// ---- VISUs/HMI.TcVIS
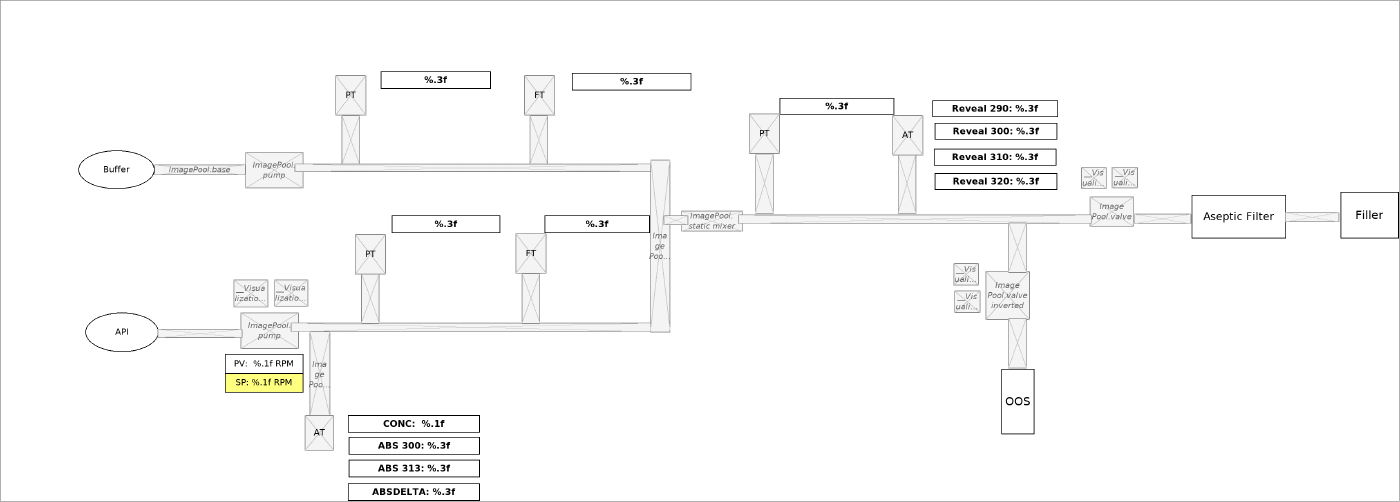
VISUALIZATION HMI  // 1787x641
    Ellipse (100,192 97x49), "Buffer"
    Ellipse (109,399 93x50), "API"
    Line (254,369)
    Line (836,413) (379,413)
    Line (449,161) (449,206)
    Line (967,273)
    Rectangle (1278,471 42x83), "OOS"
    Rectangle (1521,249 120x55), "Aseptic Filter"
    Rectangle (1711,245 74x59), "Filler"
    Image (307,399 74x46), image: ImagePool.pump
    Image (313,194 74x46), image: ImagePool.pump
    Image (869,269 79x26), image: ImagePool.static mixer
    Image (1391,251 56x38), image: ImagePool.valve
    Image (1258,346 56x62), image: ImagePool.valve inverted
    Rectangle (730,93 152x22), "%.3f", text variable: IO.FT_Buff_PV
    Rectangle (486,91 140x22), "%.3f", text variable: IO.PT_Buff_PV
    Rectangle (444,530 168x22), "CONC: %.1f", text variable: IO.AT_OPTEK_Conc_PV
    Rectangle (445,587 167x22), "ABS 313: %.3f", text variable: IO.AT_OPTEK_Abs313_PV
    Rectangle (445,558 167x22), "ABS 300: %.3f", text variable: IO.AT_OPTEK_Abs300_PV
    Rectangle (444,617 168x22), "ABSDELTA: %.3f", text variable: IO.AT_OPTEK_AbsDelta_PV
    Rectangle (500,275 138x22), "%.3f", text variable: IO.PT_API_PV
    Rectangle (695,275 134x22), "%.3f", text variable: IO.FT_API_PV
    Rectangle (995,125 146x21), "%.3f", text variable: IO.PT_PostMix_PV
    Rectangle (1190,128 160x21), "Reveal 290: %.3f", text variable: IO.AT_REVEAL_290nm_PV
    Rectangle (1193,157 156x21), "Reveal 300: %.3f", text variable: IO.AT_REVEAL_300nm_PV
    Rectangle (1192,190 156x21), "Reveal 310: %.3f", text variable: IO.AT_REVEAL_310nm_PV
    Rectangle (1193,221 156x21), "Reveal 320: %.3f", text variable: IO.AT_REVEAL_320nm_PV
    Image (676,147 23x64), image: ImagePool.pipe
    Image (436,147 23x64), image: ImagePool.pipe
    Image (371,412 464x11), image: ImagePool.base
    Image (942,274 451x11), image: ImagePool.base
    Image (376,209 461x10), image: ImagePool.base
    Image (830,204 25x220), image: ImagePool.pipe
    Image (847,275 31x12), image: ImagePool.base
    Image (197,210 116x13), image: ImagePool.base
    Image (395,423 26x110), image: ImagePool.pipe
    Image (964,196 23x77), image: ImagePool.pipe
    Image (1146,197 23x76), image: ImagePool.pipe
    Image (1287,284 23x64), image: ImagePool.pipe
    Image (1287,406 23x64), image: ImagePool.pipe
    Image (461,349 23x64), image: ImagePool.pipe
    Image (666,349 23x64), image: ImagePool.pipe
    Image (201,420 108x11), image: ImagePool.base
    Image (1447,273 73x12), image: ImagePool.base
    Image (1640,271 69x12), image: ImagePool.base
    Image (428,96 39x51), "PT", image: ImagePool.transmitter
    Image (453,299 39x51), "PT", image: ImagePool.transmitter
    Image (956,145 39x51), "PT", image: ImagePool.transmitter
    Image (658,298 39x51), "FT", image: ImagePool.transmitter
    Image (669,96 39x51), "FT", image: ImagePool.transmitter
    Image (1139,147 39x51), "AT", image: ImagePool.transmitter
    Image (389,530 37x45), "AT", image: ImagePool.inverted transmitter
    Image (298,357 44x35)
        OnMouseClick: execute { PumpsIO.P_API_START := TRUE; }
    Image (350,357 43x34)
        OnMouseClick: execute { PumpsIO.P_API_START := FALSE; }
    Rectangle (287,476 100x25), "SP: %.1f RPM", text variable: PumpsIO.SC_API_OUT
        OnMouseUp: write PumpsIO.SC_API_OUT via InputWithLimits, min 0, max 300, format %.1f
    Image (1419,213 33x27)
        OnMouseDown: execute { IO.V_FILLER_PV := FALSE; }
    Image (1380,213 32x28)
        OnMouseDown: execute { IO.V_FILLER_PV := TRUE; }
    Image (1217,336 32x28)
        OnMouseDown: execute { IO.V_OOS_PV := TRUE; }
    Image (1218,371 33x28)
        OnMouseDown: execute { IO.V_OOS_PV := FALSE; }
    Rectangle (287,452 100x25), "PV: %.1f RPM", text variable: PumpsIO.ST_API_PV
END_VISUALIZATION
